FUNCTION_BLOCK EL6070
VAR
	{attribute addProperty Name "Info data"}
	_infoData : InfoDataAds;
END_VAR

END_FUNCTION_BLOCK

(* stored: Version 1.1.0.1, ProductVersion 3.1.4024.9
   POU EL6070: Id {04c1e157-8f0f-0181-1d04-19821131d234}, SpecialFunc None *)
